TYPE ST_HeatPumpSystemEvents :
STRUCT

END_STRUCT
END_TYPE

(* stored: Version 1.1.0.1, ProductVersion 3.1.4024.12
   DUT ST_HeatPumpSystemEvents: Id {ace1aa54-0255-4ee3-acc5-c462118859e1} *)
